FUNCTION_BLOCK newProductGUIFB (* JADE WORKER *)
  (* Standard: 61499-1 *)
  (* Version 1.0, 2014-04-22, Ahmed, Fraunhofer IGD *)
  (* Compiler header: package fb.rt; *)
  (* Compiler Java Sun JDK 1.5.0 *)
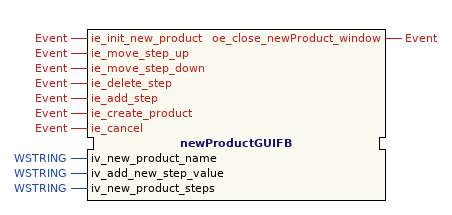
  EVENT_INPUT
    ie_init_new_product;
    ie_move_step_up;
    ie_move_step_down;
    ie_delete_step;
    ie_add_step;
    ie_create_product;
    ie_cancel;
  END_EVENT
  EVENT_OUTPUT
    oe_close_newProduct_window;
  END_EVENT
  VAR_INPUT
    iv_new_product_name : WSTRING;
    iv_add_new_step_value : WSTRING;
    iv_new_product_steps : WSTRING;
  END_VAR
END_FUNCTION_BLOCK
